# EPICS substitutions: ek9000App/Db/EL5042.substitutions
file EL5042.template
{       pattern
        {
                TERMINAL,

        }
        {
        }
}
